// TIA Portal V17 export
// export: Created 2025-06-20T10:18:27.0558345Z, ExportSetting WithDefaults, DisplayName Totally Integrated Automation Portal, DisplayVersion V17 Update 8, DisplayName TIA Portal Openness, DisplayVersion V17 Update 8, DisplayName TIA Portal Version Control Interface, DisplayVersion V17, DisplayName SINAMICS Startdrive Advanced, DisplayVersion V17 SP2, DisplayName SINAMICS Startdrive G110M, G120, G120C, G120D, G120P, G115D, DisplayVersion V17 SP2, DisplayName SINAMICS Startdrive G130, G150, S120, S150, SINAMICS MV, S210, DisplayVersion V17 SP2, DisplayName STEP 7 Professional, DisplayVersion V17 Update 8, DisplayName SINUMERIK ONE STEP 7 Toolbox, DisplayVersion V17 Update 12, DisplayName SINUMERIK ONE PLC Basic Program Plus, DisplayVersion V17 Update 12, DisplayName SINUMERIK 840D sl STEP 7 Toolbox, DisplayVersion V17 Update 12, DisplayName STEP 7 Safety, DisplayVersion V17 Update 6, DisplayName WinCC Advanced, DisplayVersion V17 Update 8
DATA_BLOCK "DB7216_RECIPES"   // DB7216
{ S7_Optimized_Access := 'FALSE'; DB_Accessible_From_OPC_UA := 'FALSE' }
AUTHOR : ETXETAR
VERSION : 1.0
// stored: AutoNumber false, DBAccessibleFromOPCUA false, DBAccessibleFromWebserver true, IsOnlyStoredInLoadMemory false, IsWriteProtectedInAS false
   VAR RETAIN
      RECIPE_NAME : Array[1..12] of Char;
      RECIPE_COUNTER_STRG : String[6] := '01';
      PART_TYPE_STRING : String[6] := '01';
      RECIPE_COUNTER : Int := 1;
      PART_TYPE_SELECTED : Int;
      PART_TYPE_INITIAL : Int := 1;
      SEQ_IN_PROCESS : Bool;   // RECIPES SEQUENCE IN PROCESS
      READY_TO_WRITE_VALUES : Bool;   // RECIPES READY TO WRITE VALUES TO CONTROL
      READING_IN_PROCESS : Bool;   // RECIPES READING IN PROCESS
      WRITING_IN_PROCESS : Bool;   // RECIPES WRITING IN PROCESS
      RECIPES_ALARM : Bool;   // RECIPES ALARM
      TIMER_RECIPES_DELAY_1 : TON_TIME;   // RECIPES DELAY 1 TIMER
      TIMER_RECIPES_DELAY_2 : TON_TIME;   // RECIPES DELAY 2 TIMER
      TIMER_RECIPES_FAULT : TON_TIME;   // RECIPES FAULT TIMER
   END_VAR
BEGIN
   RECIPE_NAME[1] := 'C';
   RECIPE_NAME[2] := 'O';
   RECIPE_NAME[3..4] := 'R';
   RECIPE_NAME[6] := '|';
   RECIPE_NAME[7] := 'T';
   RECIPE_NAME[8] := 'Y';
   RECIPE_NAME[9] := 'P';
   RECIPE_NAME[10] := 'E';
   TIMER_RECIPES_DELAY_1.PT := T#100ms;
   TIMER_RECIPES_DELAY_2.PT := T#100ms;
   TIMER_RECIPES_FAULT.PT := T#20s;
END_DATA_BLOCK
